FUNCTION EvaluateOffset : REAL
VAR_INPUT
	fRaw : REAL;				// Voltage reading (binary) from HW
END_VAR
VAR
END_VAR

EvaluateOffset := 0.0 - fRaw;

END_FUNCTION

(* stored: Version 1.1.0.1, ProductVersion 3.1.4024.15
   POU EvaluateOffset: Id {01115156-60d6-4074-8476-ab1312c666af}, SpecialFunc None *)
